// TIA Portal V20 export
FUNCTION_BLOCK "Runtime"   // FB5, LAD
{ S7_Optimized_Access := 'TRUE' }
// stored: SetENOAutomatically false
   VAR_INPUT
      "iMotor Run Freedback" : Bool;
      iTakt_1Sec : Bool;
      iReset : Bool;
      iSetTime : Bool;
   END_VAR
   VAR_IN_OUT
      ioRun_Time_C : "UDT_RunTime_Steuern";
      ioRun_Time_S : "UDT_RunTime_Status";
      "ioReset_timer-Entern" : Bool;
   END_VAR
   VAR
      sMotoris_Enabled : Bool;
      P_TRIG : Bool;
   END_VAR
   VAR_TEMP
      tVKE1 : Bool;
      tVKE0 : Bool;
   END_VAR
   VAR CONSTANT
      cCounter_PV : Int := 60;
   END_VAR
   VAR_TEMP   // added for the SCL form of the ladder/FBD networks
      _w1 : Bool;
      _w2 : Bool;
   END_VAR
BEGIN

REGION Network 1: Create tVKE1 Netzwek
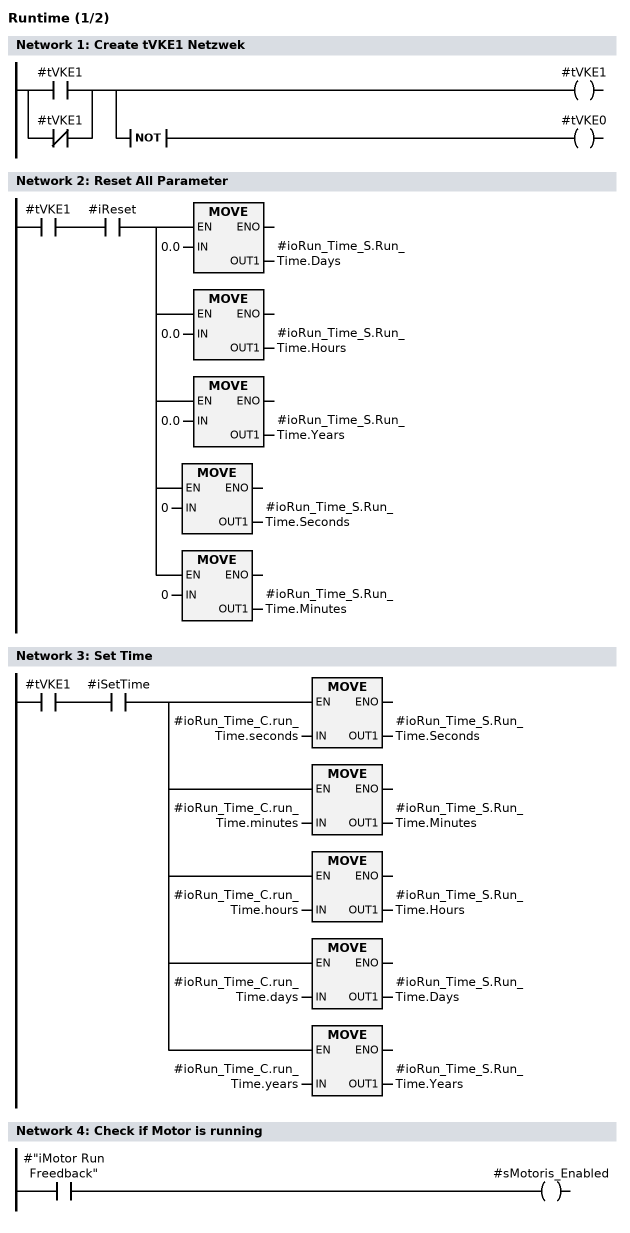
   RUNG wire#powerrail
      Contact( #tVKE1 )
      wire#w1
      Coil( #tVKE1 )
   END_RUNG
   RUNG wire#powerrail
      I_Contact( #tVKE1 )
   END_RUNG wire#w1
   RUNG wire#w1
      Not()
      Coil( #tVKE0 )
   END_RUNG
   // the same network as SCL:
   #tVKE1 := #tVKE1 OR NOT #tVKE1;
   #tVKE0 := NOT #tVKE1;
END_REGION

REGION Network 2: Reset All Parameter
   RUNG wire#powerrail
      Contact( #tVKE1 )
      Contact( #iReset )
      wire#w1
      { S7_GenerateENO := "TRUE" } Move(in := 0.0, out1 => #ioRun_Time_S.Run_Time.Days)
   END_RUNG
   RUNG wire#w1
      { S7_GenerateENO := "TRUE" } Move(in := 0.0, out1 => #ioRun_Time_S.Run_Time.Hours)
   END_RUNG
   RUNG wire#w1
      { S7_GenerateENO := "TRUE" } Move(in := 0.0, out1 => #ioRun_Time_S.Run_Time.Years)
   END_RUNG
   RUNG wire#w1
      { S7_GenerateENO := "TRUE" } Move(in := 0, out1 => #ioRun_Time_S.Run_Time.Seconds)
   END_RUNG
   RUNG wire#w1
      { S7_GenerateENO := "TRUE" } Move(in := 0, out1 => #ioRun_Time_S.Run_Time.Minutes)
   END_RUNG
   // the same network as SCL:
   IF #tVKE1 AND #iReset THEN
       #ioRun_Time_S.Run_Time.Days := 0.0;
       #ioRun_Time_S.Run_Time.Hours := 0.0;
       #ioRun_Time_S.Run_Time.Years := 0.0;
       #ioRun_Time_S.Run_Time.Seconds := 0;
       #ioRun_Time_S.Run_Time.Minutes := 0;
   END_IF;
END_REGION

REGION Network 3: Set Time
   RUNG wire#powerrail
      Contact( #tVKE1 )
      Contact( #iSetTime )
      wire#w1
      { S7_GenerateENO := "TRUE" } Move(in := #ioRun_Time_C.run_Time.seconds, out1 => #ioRun_Time_S.Run_Time.Seconds)
   END_RUNG
   RUNG wire#w1
      { S7_GenerateENO := "TRUE" } Move(in := #ioRun_Time_C.run_Time.minutes, out1 => #ioRun_Time_S.Run_Time.Minutes)
   END_RUNG
   RUNG wire#w1
      { S7_GenerateENO := "TRUE" } Move(in := #ioRun_Time_C.run_Time.hours, out1 => #ioRun_Time_S.Run_Time.Hours)
   END_RUNG
   RUNG wire#w1
      { S7_GenerateENO := "TRUE" } Move(in := #ioRun_Time_C.run_Time.days, out1 => #ioRun_Time_S.Run_Time.Days)
   END_RUNG
   RUNG wire#w1
      { S7_GenerateENO := "TRUE" } Move(in := #ioRun_Time_C.run_Time.years, out1 => #ioRun_Time_S.Run_Time.Years)
   END_RUNG
   // the same network as SCL:
   IF #tVKE1 AND #iSetTime THEN
       #ioRun_Time_S.Run_Time.Seconds := #ioRun_Time_C.run_Time.seconds;
       #ioRun_Time_S.Run_Time.Minutes := #ioRun_Time_C.run_Time.minutes;
       #ioRun_Time_S.Run_Time.Hours := #ioRun_Time_C.run_Time.hours;
       #ioRun_Time_S.Run_Time.Days := #ioRun_Time_C.run_Time.days;
       #ioRun_Time_S.Run_Time.Years := #ioRun_Time_C.run_Time.years;
   END_IF;
END_REGION

REGION Network 4: Check if Motor is running
   RUNG wire#powerrail
      Contact( #"iMotor Run Freedback" )
      Coil( #sMotoris_Enabled )
   END_RUNG
   // the same network as SCL:
   #sMotoris_Enabled := #"iMotor Run Freedback";
END_REGION

REGION Network 5: Start counting as long as Motor running
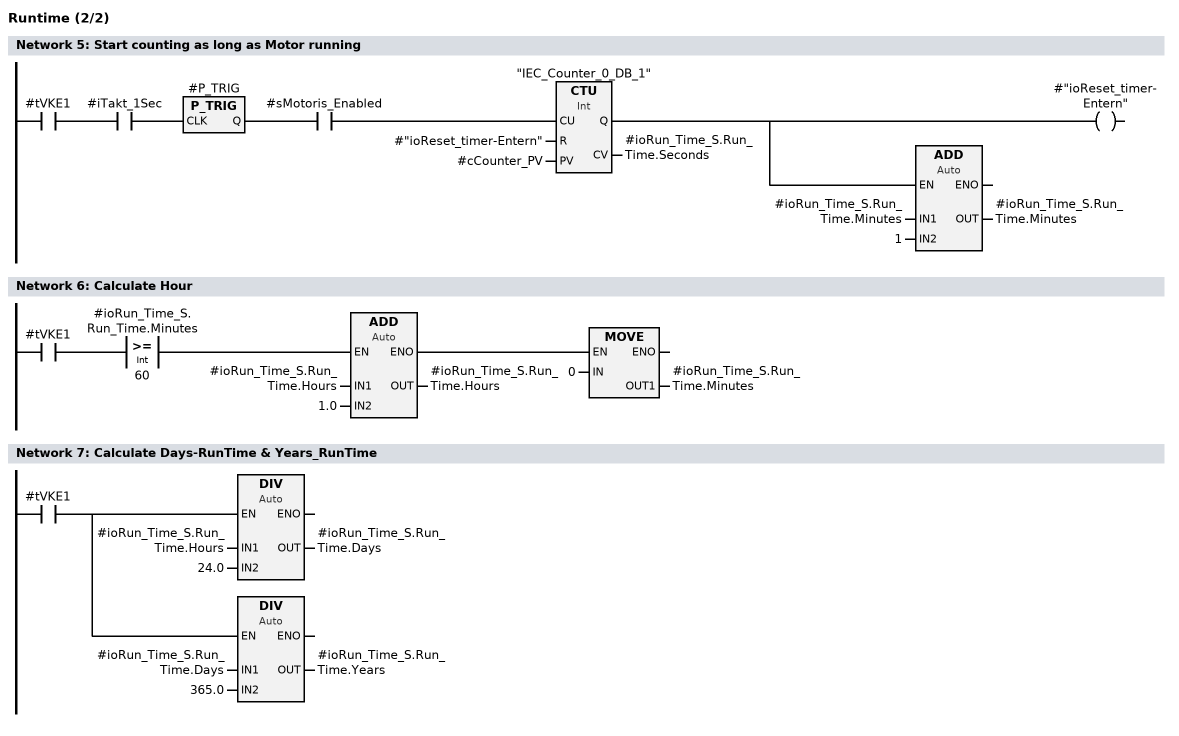
   RUNG wire#powerrail
      Contact( #tVKE1 )
      Contact( #iTakt_1Sec )
      P_Trig( #P_TRIG )
      Contact( #sMotoris_Enabled )
      { S7_Templates := "value_type := Int" } "IEC_Counter_0_DB_1".CTU(r := #"ioReset_timer-Entern", pv := #cCounter_PV, cv => #ioRun_Time_S.Run_Time.Seconds)
      wire#w1
      Coil( #"ioReset_timer-Entern" )
   END_RUNG
   RUNG wire#w1
      { S7_GenerateENO := "TRUE" } Add(in1 := #ioRun_Time_S.Run_Time.Minutes, in2 := 1, out => #ioRun_Time_S.Run_Time.Minutes)
   END_RUNG
   // the same network as SCL:
   #_w1 := #tVKE1 AND #iTakt_1Sec;
   #_w2 := #_w1 AND NOT #P_TRIG;   // rising edge
   #P_TRIG := #_w1;
   "IEC_Counter_0_DB_1".CTU(CU := #_w2 AND #sMotoris_Enabled,
                           R := #"ioReset_timer-Entern",
                           PV := #cCounter_PV,
                           CV => #ioRun_Time_S.Run_Time.Seconds);
   #"ioReset_timer-Entern" := "IEC_Counter_0_DB_1".Q;
   IF "IEC_Counter_0_DB_1".Q THEN
       #ioRun_Time_S.Run_Time.Minutes := #ioRun_Time_S.Run_Time.Minutes + 1;
   END_IF;
END_REGION

REGION Network 6: Calculate Hour
   RUNG wire#powerrail
      Contact( #tVKE1 )
      { S7_Templates := "SrcType := Int" } GE_Contact(in1 := #ioRun_Time_S.Run_Time.Minutes, in2 := 60)
      { S7_GenerateENO := "TRUE" } Add(in1 := #ioRun_Time_S.Run_Time.Hours, in2 := 1.0, out => #ioRun_Time_S.Run_Time.Hours)
      { S7_GenerateENO := "TRUE" } Move(in := 0, out1 => #ioRun_Time_S.Run_Time.Minutes)
   END_RUNG
   // the same network as SCL:
   // ENO of a box is taken as its EN; it also drops when the box reports an error
   IF #tVKE1 AND (#ioRun_Time_S.Run_Time.Minutes >= 60) THEN
       #ioRun_Time_S.Run_Time.Hours := #ioRun_Time_S.Run_Time.Hours + 1.0;
       #ioRun_Time_S.Run_Time.Minutes := 0;
   END_IF;
END_REGION

REGION Network 7: Calculate Days-RunTime & Years_RunTime
   RUNG wire#powerrail
      Contact( #tVKE1 )
      wire#w1
      { S7_GenerateENO := "TRUE" } Div(in1 := #ioRun_Time_S.Run_Time.Hours, in2 := 24.0, out => #ioRun_Time_S.Run_Time.Days)
   END_RUNG
   RUNG wire#w1
      { S7_GenerateENO := "TRUE" } Div(in1 := #ioRun_Time_S.Run_Time.Days, in2 := 365.0, out => #ioRun_Time_S.Run_Time.Years)
   END_RUNG
   // the same network as SCL:
   IF #tVKE1 THEN
       #ioRun_Time_S.Run_Time.Days := #ioRun_Time_S.Run_Time.Hours / 24.0;
       #ioRun_Time_S.Run_Time.Years := #ioRun_Time_S.Run_Time.Days / 365.0;
   END_IF;
END_REGION

REGION Network 8: End
END_REGION
END_FUNCTION_BLOCK
